// TIA Portal V19 export
DATA_BLOCK "Connect_DB"   // DB7
{ S7_Optimized_Access := 'TRUE' }
// stored: MemoryReserve 100
   VAR
      Send_C_connect { S7_SetPoint := 'True'} : TCON_Param;
      Rec_C_connect { S7_SetPoint := 'True'} : TCON_Param;
   END_VAR
BEGIN
   Send_C_connect.ID := 100;
   Send_C_connect.ACTIVE_EST := false;
   Send_C_connect.LOCAL_TSAP_ID_LEN := 2;
   Send_C_connect.REM_STADDR_LEN := 0;
   Send_C_connect.REM_TSAP_ID_LEN := 0;
   Send_C_connect.LOCAL_TSAP_ID[1] := 16#7;
   Send_C_connect.LOCAL_TSAP_ID[2] := 16#D1;
   Rec_C_connect.ID := 101;
   Rec_C_connect.ACTIVE_EST := false;
   Rec_C_connect.LOCAL_TSAP_ID_LEN := 2;
   Rec_C_connect.REM_SUBNET_ID_LEN := 0;
   Rec_C_connect.REM_STADDR_LEN := 0;
   Rec_C_connect.REM_TSAP_ID_LEN := 0;
   Rec_C_connect.LOCAL_TSAP_ID[1] := 16#7;
   Rec_C_connect.LOCAL_TSAP_ID[2] := 16#D0;
END_DATA_BLOCK
